// TIA Portal V20 export
TYPE "zmc_DatatypetoLOGS"
// stored: Access Published
   STRUCT
      Byte1 : Byte;
      Byte2 : Byte;
      Byte3 : Byte;
      Byte4 : Byte;
      Byte5 : Byte;
      Byte6 : Byte;
      Byte7 : Byte;
      Byte8 : Byte;
      Byte9 : Byte;
      Byte10 : Byte;
      Byte11 : Byte;
      Byte12 : Byte;
      Byte13 : Byte;
      Byte14 : Byte;
      Byte15 : Byte;
      Byte16 : Byte;
      Byte17 : Byte;
      Byte18 : Byte;
      DTL : DTL;
      "STRING" : String[32];
      Word1 : Word;
      Word2 : Word;
      Word3 : Word;
      Word4 : Word;
      Word5 : Word;
      Word6 : Word;
      Word7 : Word;
      Word8 : Word;
      Word9 : Word;
      Word10 : Word;
      DINT1 : DInt;
      DINT2 : DInt;
      DINT3 : DInt;
      DINT4 : DInt;
   END_STRUCT;
END_TYPE
